FUNCTION_BLOCK INTERNAL FB_StateMachine1 EXTENDS FB_StateMachine
VAR_INPUT
END_VAR
VAR_OUTPUT
END_VAR
VAR
END_VAR

END_FUNCTION_BLOCK

(* stored: Version 1.1.0.1, ProductVersion 3.1.4024.12
   POU FB_StateMachine1: Id {17d62ee0-53ef-0494-033d-53eb59531e24}, SpecialFunc None *)
